// TIA Portal V21 export
TYPE "switchgearConfig"
   STRUCT
      almMask : Word := 16#00FF;
      fbOnDelayMax : Time := T#3s;
      fbOffDelayMax : Time := T#3s;
   END_STRUCT;
END_TYPE
